FUNCTION_BLOCK lifter (* Tamplate for a simple Basic Function Block Type *)
  (* Standard: 61499-2 *)
  (* Version 0.0, 2018-01-17, 4DIAC-IDE, 4DIAC-Consortium *)
  (* Version 1.0, 2016-05-26, AZ, fortiss GmbH *)
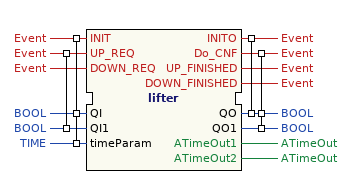
  EVENT_INPUT
    INIT WITH QI, timeParam; (* Initialization Request *)
    UP_REQ WITH QI1; (* Normal Execution Request *)
    DOWN_REQ; (* the lifter down *)
  END_EVENT
  EVENT_OUTPUT
    INITO WITH QO; (* Initialization Confirm *)
    Do_CNF WITH QO, QO1; (* Execution Confirmation *)
    UP_FINISHED;
    DOWN_FINISHED;
  END_EVENT
  VAR_INPUT
    QI : BOOL; (* Input event qualifier *)
    QI1 : BOOL; (* the value of switch *)
    timeParam : TIME;
  END_VAR
  VAR_OUTPUT
    QO : BOOL; (* Output event qualifier *)
    QO1 : BOOL; (* If UP_REQ,QO1=true; if DOWN_REQ,QO1=false *)
  END_VAR
  PLUGS
    ATimeOut1 : ATimeOut; (* time for UP *)
    ATimeOut2 : ATimeOut; (* time for down *)
  END_PLUGS
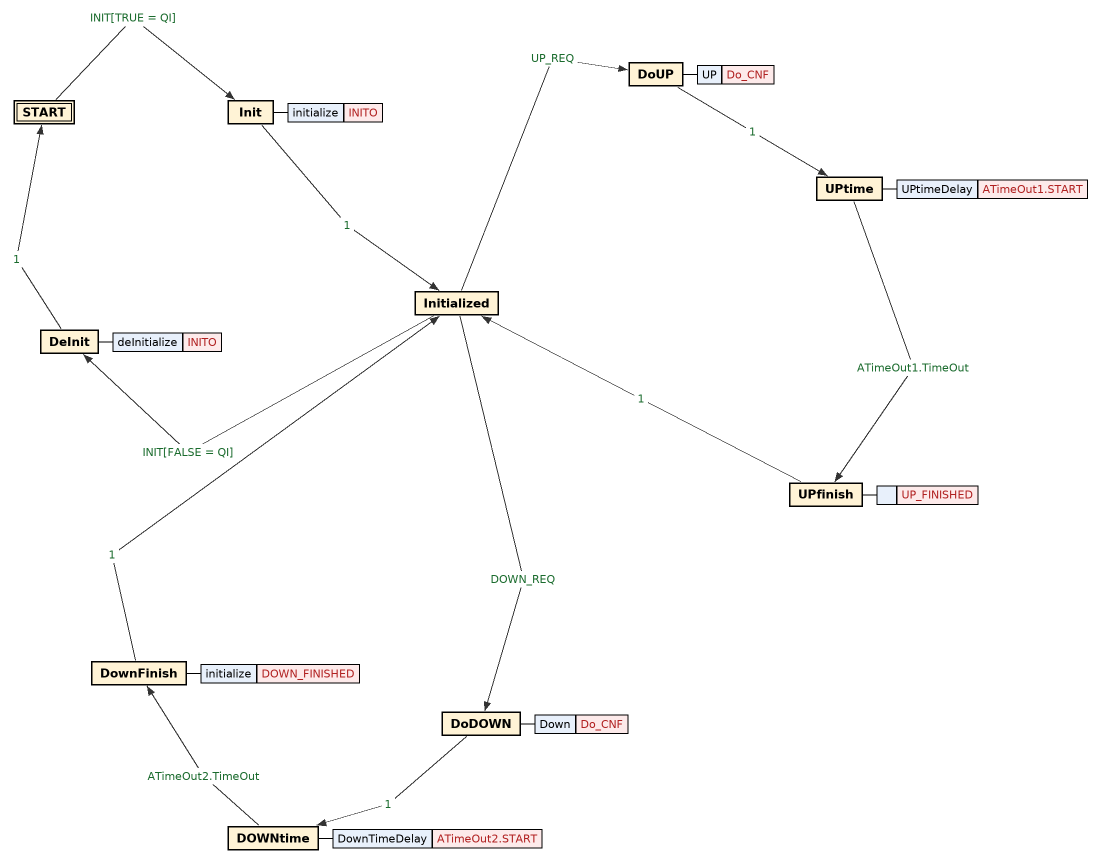
  EC_STATES
    START; (* Initial State *)
    Init : initialize -> INITO; (* Initialization *)
    DoUP : UP -> Do_CNF; (* Normal execution *)
    Initialized;
    DeInit : deInitialize -> INITO;
    UPtime : UPtimeDelay -> ATimeOut1.START;
    UPfinish : -> UP_FINISHED;
    DoDOWN : Down -> Do_CNF;
    DOWNtime : DownTimeDelay -> ATimeOut2.START;
    DownFinish : initialize -> DOWN_FINISHED;
  END_STATES
  EC_TRANSITIONS
    START TO Init := INIT[TRUE = QI];
    Init TO Initialized := 1;
    Initialized TO DoUP := UP_REQ;
    DeInit TO START := 1;
    Initialized TO DeInit := INIT[FALSE = QI];
    DoUP TO UPtime := 1;
    UPfinish TO Initialized := 1;
    Initialized TO DoDOWN := DOWN_REQ;
    DoDOWN TO DOWNtime := 1;
    DOWNtime TO DownFinish := ATimeOut2.TimeOut;
    DownFinish TO Initialized := 1;
    UPtime TO UPfinish := ATimeOut1.TimeOut;
  END_TRANSITIONS
  ALGORITHM initialize IN ST: (* Initialization algorithm *)
QO1:=FALSE;
QO := QI;
  END_ALGORITHM
  ALGORITHM deInitialize IN ST: (* Normally executed algorithm *)
QO := FALSE;
  END_ALGORITHM
  ALGORITHM UP IN ST: (* new algorithm *)
QO1:=True;
  END_ALGORITHM
  ALGORITHM UPtimeDelay IN ST: (* new algorithm *)
ATimeOut1.DT :=timeParam;
  END_ALGORITHM
  ALGORITHM Down IN ST: (* new algorithm *)
QO1:=FALSE;
  END_ALGORITHM
  ALGORITHM DownTimeDelay IN ST: (* new algorithm *)
ATimeOut2.DT:= timeParam;
  END_ALGORITHM
END_FUNCTION_BLOCK
